{attribute addProperty BoxType "EL3423-0000-0020"}
{attribute addProperty Id "Reactive_EnergyAT %I*LINT648"}
{attribute addProperty CRC "2842626133"}
{attribute addProperty SizeInBites "64"}
{attribute addProperty SizeInBytes "8"}
TYPE Total_Reactive_Reduced_A96F0855 :
STRUCT
	{attribute addProperty Name "Reactive_Energy"}
	Reactive_Energy AT %I* : LINT;
END_STRUCT
END_TYPE

(* stored: Version 1.2.0.0, ProductVersion 3.1.4024.9
   DUT Total_Reactive_Reduced_A96F0855: Id {fe7babc4-4856-4ee4-a7dc-2f6f35e269db} *)
